{attribute 'qualified_only'}
TYPE E_HMI_DriveStatus :
(
	UNKNOWN := 0,
	STOPPED := 1,
	RUNNING := 2,
	ERROR 	:= 3
);
END_TYPE

(* stored: Version 1.1.0.1
   DUT E_HMI_DriveStatus: Id {30a76562-a2f9-4391-ad18-830ee7c84e54} *)
